FUNCTION_BLOCK FB_Transport_A
VAR_INPUT
	bStop1 :BOOL;
	bStop2 :BOOL;
	bStop3 :BOOL;
END_VAR
VAR_OUTPUT
	//Hardware Outputs
	bStopper1 :BOOL;
	bStopper2 :BOOL;
	bStopper3 :BOOL;
END_VAR
VAR
END_VAR

bStopper1 :=bStop1;
bStopper2 :=bStop2;
bStopper3 :=bStop3;

END_FUNCTION_BLOCK

(* stored: Version 1.1.0.1, ProductVersion 3.1.4024.15
   POU FB_Transport_A: Id {92d8dfbb-6f4b-4a1d-b043-07c429309538}, SpecialFunc None *)
